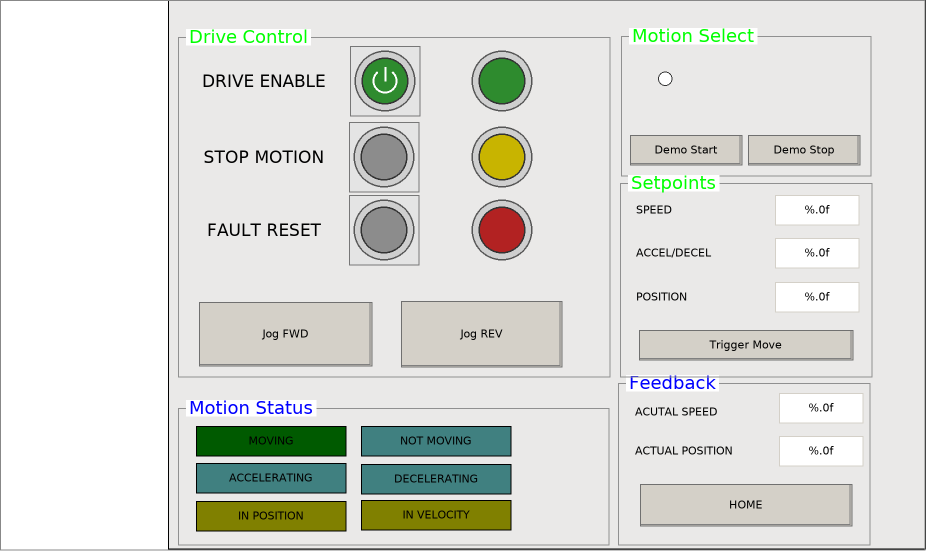
VISUALIZATION MotorFaceplate  // 926x551
    Rectangle (168,-2 758x551)
    GroupBox (178,29 432x348), "Drive Control"
        PowerSwitch (172,17 70x70), variable: gvlServo.servo1Interface.bDriveEnable, behaviour: TOGGLE, style: Switch-PowerSwitch-Green
        PushSwitch (171,93 70x70), variable: gvlServo.servo1Interface.bStopMotion, behaviour: TAP, style: Switch-PushSwitch-Gray
        PushSwitch (171,166 70x70), variable: gvlServo.servo1Interface.bFaultReset, behaviour: TAP, style: Switch-PushSwitch-Gray
        Lamp1 (289,17 70x70), variable: gvlServo.servo1Interface.bDriveEnabled, style: Lamp-Lamp1-Green
        Lamp1 (289,93 70x70), variable: gvlServo.servo1Interface.bNotMoving, style: Lamp-Lamp1-Yellow
        Lamp1 (289,166 70x70), variable: gvlServo.servo1Interface.bFaulted, style: Lamp-Lamp1-Red
        Label (11,37 150x30), "DRIVE ENABLE"
        Label (11,113 150x30), "STOP MOTION"
        Label (11,186 150x30), "FAULT RESET"
        Button (21,273 173x64), "Jog FWD"
            tap gvlServo.servo1Interface.bJogFWD
        Button (223,272 161x66), "Jog REV"
            tap gvlServo.servo1Interface.bJogRev
    GroupBox (178,400 431x145), "Motion Status"
        RoundedRectangle (18,26 150x30), "MOVING", colour toggle: gvlServo.servo1Interface.bMoving
        RoundedRectangle (183,26 150x30), "NOT MOVING", colour toggle: gvlServo.servo1Interface.bNotMoving
        RoundedRectangle (18,63 150x30), "ACCELERATING", colour toggle: gvlServo.servo1Interface.bAccelerating
        RoundedRectangle (183,64 150x30), "DECELERATING", colour toggle: gvlServo.servo1Interface.bDecelerating
        RoundedRectangle (18,101 150x30), "IN POSITION", colour toggle: gvlServo.servo1Interface.bInposition
        RoundedRectangle (183,100 150x30), "IN VELOCITY", colour toggle: gvlServo.servo1Interface.bInVelocity
    GroupBox (618,375 252x170), "Feedback"
        Textfield (161,18 84x30), "%.0f", text variable: gvlServo.servo1Interface.rActualSpeed
        Label (14,61 120x30), "ACTUAL POSITION"
        Textfield (161,61 84x30), "%.0f", text variable: gvlServo.servo1Interface.rActualPosition
        Label (14,22 108x30), "ACUTAL SPEED"
        Button (22,109 212x42), "HOME", invisible if: TRUE
            tap gvlServo.servo1Interface.bHome
    GroupBox (621,28 250x148), "Motion Select"
        RadioButton (35,21 173x59), variable: gvlServo.servo1Interface.iMotionSelect
            p3123465237: DEMO MODE
            p2481256679: RELATIVE POSITION
            p1032612214: VELOCITY CONTROL
        Button (9,107 112x30), "Demo Start", invisible if: gvlServo.servo1Interface.iMotionSelect = 0
            tap gvlServo.servo1Interface.bDemoModeStart
        Button (127,107 112x30), "Demo Stop", invisible if: gvlServo.servo1Interface.iMotionSelect = 0
            tap gvlServo.servo1Interface.bDemoModeStop
    GroupBox (620,175 252x202), "Setpoints"
        Label (13,20 76x30), "SPEED", invisible if: TRUE
        Textfield (155,20 84x30), "%.0f", text variable: gvlServo.servo1Interface.rSpeed, invisible if: TRUE
        Label (13,63 99x30), "ACCEL/DECEL", invisible if: TRUE
        Textfield (155,63 84x30), "%.0f", text variable: gvlServo.servo1Interface.rAccelDecel, invisible if: TRUE
        Label (13,107 76x30), "POSITION", invisible if: TRUE
        Textfield (155,107 84x30), "%.0f", text variable: gvlServo.servo1Interface.rPosition, invisible if: TRUE
        Button (19,155 214x30), "Trigger Move", invisible if: TRUE
            tap gvlServo.servo1Interface.bTriggerMove
END_VISUALIZATION

(* stored: Version 1.1.0.1, ProductVersion 3.1.4024.12
   Visu MotorFaceplate: Id {bc574e3f-2d19-4968-ab47-e788405f6744} *)
